{attribute 'qualified_only'}
{attribute 'strict'}
TYPE E_STATION_STATE :
(
	uninit,
	idle,
	do_action1,
	do_action2,
	do_action3,
	do_action4,
	do_action5,
	do_action6,
	do_action7,
	do_action8,
	do_action9,
	done,
	pause,
	error
);
END_TYPE

(* stored: Version 1.1.0.1, ProductVersion 3.1.4024.12
   DUT E_STATION_STATE: Id {82c78350-fa63-4bdf-bd73-d1b280128060} *)
